PROGRAM prgGrid
VAR
	fbGrid					: FB_Grid_Power;
	fbCounter				: FB_EnergyCounter;
	lrGridPower				: LREAL;	//{#lynus.ag#()}
	byErrorWarningGrid		: BYTE;		//{#lynus.ag#()}
END_VAR
VAR PERSISTENT
	rSizeGrid				: REAL;		//{#lynus.ag#()}
	lrCounterGridCons		: LREAL;	//{#lynus.ag#()}
	lrCounterGridProd		: LREAL;	//{#lynus.ag#()}
END_VAR

fbGrid(
	bEnable:= TRUE, 
	diNrOfEMS_IN:= prgEMS.EMS.diNrOfEMS_OUT, 
	diNrOfEM_IN_Grid:= prgXelect.fbBatt.diNrOfEM_OUT_Grid, 
	rSizeGridConn:= rSizeGrid, 
	stDataGrid=> , 
	diNrOfGrid_OUT=> );
	
lrGridPower := fbGrid.stDataGrid.lrPower;
byErrorWarningGrid := fbGrid.stDataGrid.byErrorWarning;

fbCounter(
	byActiveTariff:= 1, 
	lrPowerInput:= lrGridPower, 
	lrTotalCounterEnergy_Consumption=> , 
	lrTotalCounterEnergy_Production=> , 
	lrCounterEnergyT1_Consumption=> , 
	lrCounterEnergyT2_Consumption=> , 
	lrCounterEnergyT1_Production=> , 
	lrCounterEnergyT2_Production=> );

IF fbCounter.lrTotalCounterEnergy_Consumption > lrCounterGridCons THEN
	lrCounterGridCons := fbCounter.lrTotalCounterEnergy_Consumption;
END_IF
	IF fbCounter.lrTotalCounterEnergy_Production > lrCounterGridProd THEN
		lrCounterGridProd := fbCounter.lrTotalCounterEnergy_Production;
	END_IF

END_PROGRAM

(* stored: Version 1.1.0.1, ProductVersion 3.1.4024.9
   POU prgGrid: Id {34200d71-fb30-4541-aed0-759ca7d5cb5d}, SpecialFunc None *)
